SUBAPPLICATION Uebung_035a1b_AX (* Ampelsteuerung mit Pattern Sequencer (AX) und Bit-Assembler *)
  (* Standard: 61499-2; Description: Copyright (c) 2023 Meisterschulen am Ostbahnhof This program and the accompanying materials are made available under the terms of the Eclipse Public License 2.0 which is available at https://www.eclipse.org/legal/epl-2.0/ SPDX-License-Identifier: EPL-2.0 *)
  (* Version 1.0, 2026-02-01, Franz Höpfinger, Meisterschulen am Ostbahnhof, initial API and implementation and/or initial documentation *)
  PACKAGE Uebungen;
  IMPORT logiBUS::io::DI::logiBUS_DI::Input_I1;
  IMPORT logiBUS::io::DI::logiBUS_DI_Events::BUTTON_SINGLE_CLICK;
  IMPORT logiBUS::io::DQ::logiBUS_DO::Output_Q1;
  IMPORT logiBUS::io::DQ::logiBUS_DO::Output_Q2;
  IMPORT logiBUS::io::DQ::logiBUS_DO::Output_Q3;
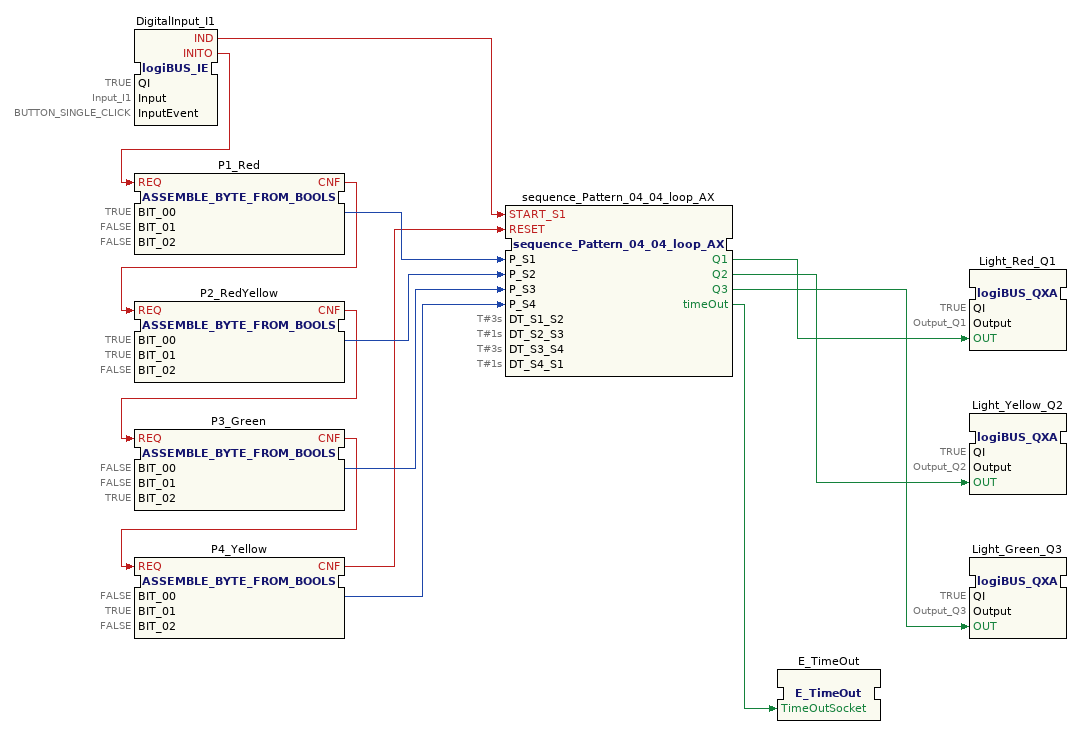
  FBS
    sequence_Pattern_04_04_loop_AX : logiBUS::utils::sequence::pattern::sequence_Pattern_04_04_loop_AX(DT_S1_S2 := T#3s, DT_S2_S3 := T#1s, DT_S3_S4 := T#3s, DT_S4_S1 := T#1s);
    DigitalInput_I1 : logiBUS::io::DI::logiBUS_IE(QI := TRUE, Input := Input_I1, InputEvent := BUTTON_SINGLE_CLICK);
    Light_Red_Q1 : logiBUS::io::DQ::logiBUS_QXA(QI := TRUE, Output := Output_Q1);
    Light_Yellow_Q2 : logiBUS::io::DQ::logiBUS_QXA(QI := TRUE, Output := Output_Q2);
    Light_Green_Q3 : logiBUS::io::DQ::logiBUS_QXA(QI := TRUE, Output := Output_Q3);
    P1_Red : eclipse4diac::utils::assembling::ASSEMBLE_BYTE_FROM_BOOLS(BIT_00 := TRUE (* RED *), BIT_01 := FALSE (* YELLOW *), BIT_02 := FALSE (* GREEN *));
    P2_RedYellow : eclipse4diac::utils::assembling::ASSEMBLE_BYTE_FROM_BOOLS(BIT_00 := TRUE (* RED *), BIT_01 := TRUE (* YELLOW *), BIT_02 := FALSE (* GREEN *));
    P3_Green : eclipse4diac::utils::assembling::ASSEMBLE_BYTE_FROM_BOOLS(BIT_00 := FALSE (* RED *), BIT_01 := FALSE (* YELLOW *), BIT_02 := TRUE (* GREEN *));
    P4_Yellow : eclipse4diac::utils::assembling::ASSEMBLE_BYTE_FROM_BOOLS(BIT_00 := FALSE (* RED *), BIT_01 := TRUE (* YELLOW *), BIT_02 := FALSE (* GREEN *));
    E_TimeOut : iec61499::events::E_TimeOut;
  END_FBS
  EVENT_CONNECTIONS
    DigitalInput_I1.IND TO sequence_Pattern_04_04_loop_AX.START_S1;
    DigitalInput_I1.INITO TO P1_Red.REQ;
    P1_Red.CNF TO P2_RedYellow.REQ;
    P2_RedYellow.CNF TO P3_Green.REQ;
    P3_Green.CNF TO P4_Yellow.REQ;
    P4_Yellow.CNF TO sequence_Pattern_04_04_loop_AX.RESET;
  END_CONNECTIONS
  DATA_CONNECTIONS
    P1_Red. TO sequence_Pattern_04_04_loop_AX.P_S1;
    P2_RedYellow. TO sequence_Pattern_04_04_loop_AX.P_S2;
    P3_Green. TO sequence_Pattern_04_04_loop_AX.P_S3;
    P4_Yellow. TO sequence_Pattern_04_04_loop_AX.P_S4;
  END_CONNECTIONS
  ADAPTER_CONNECTIONS
    sequence_Pattern_04_04_loop_AX.Q1 TO Light_Red_Q1.OUT;
    sequence_Pattern_04_04_loop_AX.Q2 TO Light_Yellow_Q2.OUT;
    sequence_Pattern_04_04_loop_AX.Q3 TO Light_Green_Q3.OUT;
    sequence_Pattern_04_04_loop_AX.timeOut TO E_TimeOut.TimeOutSocket;
  END_CONNECTIONS
END_SUBAPPLICATION
